// TIA Portal V18 export
// export: Created 2025-12-01T12:37:59.8609871Z, ExportSetting None, DisplayName Totally Integrated Automation Portal, DisplayVersion V18 Update 5, DisplayName TIA Portal Openness, DisplayVersion V18 Update 5, DisplayName TIA Portal Teamcenter Gateway, DisplayVersion V18, DisplayName TIA Portal Version Control Interface, DisplayVersion V18, DisplayName STEP 7 Professional, DisplayVersion V18 Update 5, DisplayName STEP 7 Safety, DisplayVersion V18, DisplayName WinCC Professional, DisplayVersion V18 Update 5
FUNCTION "Diagnostic" : Void   // FC3001, SCL
TITLE = Diagnostic
{ S7_Optimized_Access := 'FALSE' }
AUTHOR : STD
FAMILY : RCS
VERSION : 18.0
// stored: AutoNumber false, SetENOAutomatically true
   VAR_INPUT
      iCPUType : Int;   // 1-DP&PN 2-PN
      iDBNum : Word;
      iOffset : Int;   // Start address
      iHardwareID : HW_IOSYSTEM;
   END_VAR
   VAR_OUTPUT
      oStatus : Int;
   END_VAR
   VAR_TEMP
      RDSRet : Struct
         Busy : Bool;
         Header : Struct
            Length : Word;
            Number : Word;
         END_STRUCT;
      END_STRUCT;
      retInt : Int;
      SSL : Struct
         SSID : Word;
         Index : Word;
         Length : Int;
      END_STRUCT;
      DR : Any;
      DRS AT DR : Struct
         SyntaxID : Byte;
         DataType : Byte;
         RepetitionFactor : Int;
         DB_Number : Word;
         MemoryAreaAddress : DWord;
      END_STRUCT;
   END_VAR
BEGIN

   (*############################################################
      RUHLAMAT SUZHOU ELEC.STD.
      Copyright (c) 2017. All rights reserved.    

      NAME OF FUNCTION BLOCK:         Diagnostic
      VERSION NUMBER:                 V3.0
      COMPOSER:                       Ming.Jiang

      CreateDate:                    16.Nov.2016
      ----------------------------------------------------------
      Interface description:
      IN:
          "iCPUType"
          iDBNum
          iOffset
          iHardwareID

      INOUT:
      OUT:
          oStatus

      ----------------------------------------------------------
      #RET_VALUE:

      #Alert Value:

      ----------------------------------------------------------
      Date           Name      Version           Activity                                                                              
      28.Nov.2016    JM        V3.0              add alarm

   ############################################################*)
   IF #iCPUType = 0 OR #iDBNum = 0 THEN
       ENO := 0;
       RETURN;
   ELSE
       IF #iCPUType=2 THEN
           GOTO PN;
       ELSIF #iCPUType=1 THEN
           ;
       ELSE
           ENO := 0;
           RETURN;
       END_IF;
       #DRS.SyntaxID := 16#10;
       #DRS.DataType := 16#02;
       #DRS.RepetitionFactor := 128;
       #DRS.DB_Number := #iDBNum;
       #DRS.MemoryAreaAddress := 16#8400_0000 OR (SHL(IN := INT_TO_DWORD(#iOffset), N := 3));
       #oStatus := DeviceStates(LADDR := #iHardwareID, MODE := 2, STATE := #DR);
   PN:
       #DRS.SyntaxID := 16#10;
       #DRS.DataType := 16#02;
       #DRS.RepetitionFactor := 128;
       #DRS.DB_Number := #iDBNum;
       #DRS.MemoryAreaAddress := 16#8400_0000 OR (SHL(IN := INT_TO_DWORD(#iOffset), N := 3));
       #oStatus := DeviceStates(LADDR := #iHardwareID, MODE := 2, STATE := #DR);
       // orginise interface data 
       ENO := 1;
       RETURN;
   END_IF;
END_FUNCTION
